// TwinCAT 3 PLC project Untitled1
// ProgramVersion: 3.1.4024.0
// libraries:
//   Tc2_Standard, * (Beckhoff Automation GmbH)
//   Tc2_System, * (Beckhoff Automation GmbH)
//   Tc3_Module, * (Beckhoff Automation GmbH)
// project tree:
//   GVLs/ GVL.TcGVL (not stored)
//   POUs/ GetWaterDuration.TcPOU, MonitoringTheSoilTask.TcPOU, WateringTask.TcPOU
//   VISUs/ PlcTask.TcTTO, Task_4.TcTTO, Task_5.TcTTO

CONFIGURATION Untitled1
    RESOURCE PLC ON TwinCAT3
        TASK PlcTask(INTERVAL := T#10ms, PRIORITY := 20);
        TASK Task_4(INTERVAL := T#10ms, PRIORITY := 1);
        TASK Task_5(INTERVAL := T#10ms, PRIORITY := 2);
        PROGRAM MonitoringTheSoilTask WITH PlcTask : MonitoringTheSoilTask;
        PROGRAM WateringTask WITH Task_4 : WateringTask;
    END_RESOURCE
END_CONFIGURATION

// ---- POUs/MonitoringTheSoilTask.TcPOU
PROGRAM MonitoringTheSoilTask
VAR
	Timer: TON;
	state: INT;
	Moisture: REAL;
	Temp: REAL;
	WaterRequired: BOOL;
END_VAR

CASE state OF
	0:// Initial position
	Moisture :=50;
	Temp := 25;
	state :=1;
	
	1: //ReadSensors
	Moisture:= Moisture - 1;
	IF Moisture < 0 THEN Moisture :=0 ;END_IF;
	Temp := Temp;
	state := 2;
	 
	2://UpdateGVL
	WaterRequired := (Moisture <30 AND Temp > 20 );
	State:=1;

	
	
	
	
END_CASE

END_PROGRAM

// ---- POUs/WateringTask.TcPOU
PROGRAM WateringTask
VAR
	WaterTimer:TON;
	Delay:TON;
	state:INT;
	Moisture: REAL;
	Temp: REAL;
	WaterRequired: BOOL;
END_VAR

 	
//Watering control
CASE state OF
	
	
	0:// Initial position
	gvl.WaterON:= FALSE;
	state:=1;
	1:// Checking the conditions
	IF gvl.WaterRequired THEN
				gvl.WaterDuration := GetWaterDuration(gvl.Moisture, Temp);
				gvl.WaterON := TRUE;	
				WaterTimer(IN := TRUE, PT := gvl.WaterDuration);
				State := 2;
			ELSE
				State := 3;
			END_IF;
			
	2:  // Watering
	WaterTimer(IN := TRUE);
			IF WaterTimer.Q THEN
			  gvl.WaterON := FALSE;
	GVL.WaterRequired := FALSE;
	END_IF
	WaterTimer(IN := FALSE);
				state := 3;
	3:// Idle
	Delay(IN:=TRUE, PT:=T#5S);
	IF NOT(Delay.Q) THEN
		RETURN;
	END_IF
	Delay(In:=FALSE);
	state:=1;		
END_CASE

END_PROGRAM

// ---- POUs/GetWaterDuration.TcPOU
FUNCTION GetWaterDuration : TIME
VAR_INPUT
	MoistIn:REAL ;
	TempIn:REAL;
END_VAR
VAR
	rSeconds : REAL; 
    udiMs : UDINT; // milliseconds as unsigned integer
END_VAR

// Calculate duration in seconds
rSeconds := 10.0 + (TempIn - 20.0) - (MoistIn * 0.1);

// Convert to ms, then to UDINT
udiMs := LREAL_TO_UDINT(REAL_TO_LREAL(rSeconds) * 1000.0);

// Convert to TIME
GetWaterDuration := UDINT_TO_TIME(udiMs);

// Clamp between 5s and 30s
IF GetWaterDuration < T#5s THEN GetWaterDuration := T#5s; END_IF;
IF GetWaterDuration > T#30s THEN GetWaterDuration := T#30s; END_IF;

END_FUNCTION
